// TwinCAT 3 PLC project PLCPro
// ProgramVersion: 3.1.4024.0
// libraries:
//   Tc2_Standard, * (Beckhoff Automation GmbH)
//   Tc2_System, * (Beckhoff Automation GmbH)
//   Tc2_Utilities, * (Beckhoff Automation GmbH)
//   Tc3_IotBase, * (Beckhoff Automation GmbH)
//   Tc3_JsonXml, * (Beckhoff Automation GmbH)
//   Tc3_Module, * (Beckhoff Automation GmbH)
// project tree:
//   / PlcTask.TcTTO
//   POUs/ MockServer.TcPOU, MAIN.TcPOU, EtonSmartBreaker.TcPOU, PostmanEco.TcPOU
// real-time tasks:
//   TASK PlcTask: cycle T#10ms, priority 20, ADS port 350

CONFIGURATION PLCPro
    RESOURCE PLC ON TwinCAT3
        TASK PlcTask(INTERVAL := T#10ms, PRIORITY := 20);
        PROGRAM MAIN WITH PlcTask : MAIN;
    END_RESOURCE
END_CONFIGURATION

// ---- POUs/MAIN.TcPOU
PROGRAM MAIN
VAR
	//Client
	//fbhttpClient : FB_IotHttpClient := (sHostName:='postman-echo.com',
	//							  	bKeepAlive:=TRUE, tConnectionTimeout:=T#10S);
									
	//Eton
	fbhttpClient : FB_IotHttpClient := (sHostName:='api.em.eaton.com',
								  	bKeepAlive:=TRUE, tConnectionTimeout:=T#10S);		
				
	//Get Request
	fbRequest : FB_IotHttpRequest;		
	state : (IDLE, SEND_REQUEST, WAIT_FOR_RESPONSE, READ_RESPONSE,ERROR,FORMATER);			
	sendGetRequest: BOOL;
	debugContent : STRING(511);
	fbJsonParser : FB_JsonDomParser;
	jsonDoc				: SJsonValue;
	jsonArgsMember				: SJsonValue;
	jsonFoo2 : SJsonValue;
	results : STRING;
	
	//JSON Formater
	fbJsonWriter         : FB_JsonSaxWriter;
	sendData                : STRING(2000);
	
END_VAR

//PostmanEco();
MockServer();
//EtonSmartBreaker();

END_PROGRAM

// ---- POUs/MockServer.TcPOU
PROGRAM MockServer
VAR
	//Mock Server
	fbhttpClient : FB_IotHttpClient := (sHostName:='4446f140-18dd-4b14-8279-3cc341a02b1e.mock.pstmn.io',
								  	bKeepAlive:=TRUE, tConnectionTimeout:=T#10S);		
				
	//Get Request
	fbRequest : FB_IotHttpRequest;		
	state : (IDLE, SEND_REQUEST, WAIT_FOR_RESPONSE, READ_RESPONSE,ERROR,HEADER);			
	sendGetRequest: BOOL;
	debugContent : STRING(511);
	fbJsonParser : FB_JsonDomParser;
	jsonDoc				: SJsonValue;
	jsonArgsMember				: SJsonValue;
	jsonMachineName : SJsonValue;
	results : STRING;
	
	//Header
	fbHeaderField : FB_IotHttpHeaderFieldMap;
END_VAR

// Init client parameters at startup
IF NOT fbhttpClient.bConfigured THEN 
	fbhttpClient.nHostPort:= 443; //80 for http  443 For https
	fbhttpClient.stTLS.bNoServerCertCheck:= TRUE;
END_IF

	
//Get Request
CASE state OF
	
	//Send Get Request
	IDLE:
		IF sendGetRequest THEN
			state := HEADER;
			sendGetRequest := FALSE;
		END_IF
	
	//Create Autorization Header File
	HEADER:
		fbHeaderField.AddField(sField:='Header1',sValue:='1',bAppendValue:=FALSE);
		fbHeaderField.AddField(sField:='Header2',sValue:='2',bAppendValue:=FALSE);
		state := SEND_REQUEST;
	
	//Send Get Request
	SEND_REQUEST:                                                                                      
		IF fbRequest.SendRequest(sUri:='/getmockdata', 
			fbClient:=fbhttpClient, eRequestType:=ETcIotHttpRequestType.HTTP_Get, 
				0, 0,fbHeader:=fbHeaderField ) THEN
			state := WAIT_FOR_RESPONSE;
		END_IF
	
	//Wait for Response
	WAIT_FOR_RESPONSE:

		IF NOT fbRequest.bBusy THEN
			IF fbRequest.bError THEN
				state := ERROR;
			ELSE
				state := READ_RESPONSE;
			END_IF
		END_IF
	
	//Read Response	
	READ_RESPONSE:
	
		//Get Response Content
		fbRequest.GetContent(pContent:= ADR(debugContent), nContentSize:= SIZEOF(debugContent), bSetNullTermination:= TRUE);
		
		//Check Status 
		IF fbRequest.nStatusCode >= 200 AND fbRequest.nStatusCode < 300 THEN
			jsonDoc:= fbRequest.GetJsonDomContent(fbJsonParser);
			
			//Check response has data in body
			IF jsonDoc <> 0 THEN
				
				//Check machine key is present 
				IF fbJsonParser.HasMember(jsonDoc, 'machine') THEN
					
					//Get Value for the specifed key
					jsonArgsMember:= fbJsonParser.FindMember(jsonDoc, 'machine');
					
					//Check wether data has an name key 	
					IF fbJsonParser.HasMember(jsonArgsMember, 'name')  THEN
						
						//Get Value for the specifed key
						jsonMachineName:= fbJsonParser.FindMember(jsonArgsMember, 'name');
						
							//Check data is a String
							IF fbJsonParser.IsString(jsonMachineName) THEN	
								
								//Get the Data 		
								results:= fbJsonParser.GetString(jsonMachineName);									
							END_IF
					END_IF
				END_IF
			END_IF
		END_IF
		state := IDLE;
		
	ERROR:
		//
		
		
END_CASE

//Cyclic Client 
fbhttpClient.Execute();

END_PROGRAM

// ---- POUs/EtonSmartBreaker.TcPOU
PROGRAM EtonSmartBreaker
VAR
	//Eaton Server
	fbhttpClient : FB_IotHttpClient := (sHostName:='api.em.eaton.com',
								  	bKeepAlive:=TRUE, tConnectionTimeout:=T#10S);		
	
	//Get Request
	fbRequest : FB_IotHttpRequest;		
	state : (IDLE, SEND_REQUEST, WAIT_FOR_RESPONSE, READ_RESPONSE,ERROR,ADD_HEADER);			
	sendGetRequest: BOOL;
	debugContent : STRING(2000);
	fbJsonParser : FB_JsonDomParser;
	jsonDoc				: SJsonValue;
	jsonArgsMember				: SJsonValue;
	jsonMachineName : SJsonValue;
	results : STRING;
	
	//Header
	fbHeaderField : FB_IotHttpHeaderFieldMap;
	sAuthoToken : STRING(2000);
END_VAR

// Init client parameters at startup
IF NOT fbhttpClient.bConfigured THEN 
	fbhttpClient.nHostPort:= 443; //80 for http  443 For https
	fbhttpClient.stTLS.bNoServerCertCheck:= TRUE;
END_IF

	
//Get Request
CASE state OF
	
	//Send Get Request
	IDLE: 
		IF sendGetRequest THEN
			state := ADD_HEADER;
			sendGetRequest := FALSE;
		END_IF
	
	//Create Autorization Header File
	ADD_HEADER:
		sAuthoToken := 'Bearer eyJraWQiOiJFZHViWGxfQVg2emd3R044b0dOa21VRUxRWHEyOUdOQzNJUjFrcFdtVGZBIiwiYWxnIjoiUlMyNTYifQ.eyJ2ZXIiOjEsImp0aSI6IkFULjhjYU5jckV2aU56UHBKNEk1bEQ2YVh0amxjVTJ2TG9xQ29wcmNWd0ExdVUiLCJpc3MiOiJodHRwczovL2lkLmVhdG9uLmNvbS9vYXV0aDIvYXVzOWQ4dnhlOFZNWTFod0M0eDciLCJhdWQiOiJhcGk6Ly9ibGMiLCJpYXQiOjE3Mjc5MzE0MjMsImV4cCI6MTcyNzkzNTAyMywiY2lkIjoiMG9hbTgzZHR2dVdnV1FTNjk0eDciLCJzY3AiOlsiY2xpZW50X2NyZWQiXSwiYWRvcHRlcmlkIjoiYjgzYjJlZjItMmJhZi1iZTEzLTNmOGItZGI3ZmQyNWYyMDE3Iiwic3ViIjoiMG9hbTgzZHR2dVdnV1FTNjk0eDciLCJibGNzYWlkIjoiMGEzYmVhYTctZTE1ZS00N2U1LTlhMmItY2ZjYjE3ZGU1ZDQ0IiwibmFtZSI6IiAifQ.00_Ss224pRcBLPLgnpvzWnFV0GmS_tGB9qeZJu8OeWvd7kSRdSMygCW7wede4vqgu5Ubb5BiEe9cokUyDZlxNh-5BjZUgMOYV3XZXAJ5Rhxdnk4yjf6ERhz2HZ8PuB8aCMRdxaAe6N6f_PemYtNiTWQ7DWPPc7aFGsk2gy1FRxRTvX5XlgX2cIQoJKBBEq6lzWZOUW8Jl9Aw2f90uQ6BSJRAfazYmr6yWAjuQoOGHQlXHmZxGf1fEm9NqKGUeh5tYEAE-YueOLzh__bxsjUHR1NJwBrpN3sa3_VFoNzfGEunkiQ1RyFZyzoUS3xEB2QbCjJTgo47z_0nJobPwB3EDg';
		fbHeaderField.AddField(sField:='Em-Api-Subscription-Key',sValue:='666585a90d81461da51fb9ed6fa14c7b',bAppendValue:=FALSE);
		fbHeaderField.AddField(sField:='Authorization',sValue:=sAuthoToken,bAppendValue:=FALSE);
		//fbHeaderField.AddField(sField:='Accept',sValue:='application/json',bAppendValue:=FALSE);
		//fbHeaderField.AddField(sField:='Content-Type',sValue:='application/json',bAppendValue:=FALSE);
		//fbHeaderField.AddField(sField:='Cache-Control',sValue:='no-cache',bAppendValue:=FALSE);
		//fbHeaderField.AddField(sField:='Connection',sValue:='keep-alive',bAppendValue:=FALSE);
		state := SEND_REQUEST;
	
	//Send Get Request
	SEND_REQUEST:                                                                             
		IF fbRequest.SendRequest(sUri:='/api/v1/devices/c595f832-81c8-44c9-ba4a-0b3c9b980dc4/breaker/remoteHandle/position', 
			fbClient:=fbhttpClient, eRequestType:=ETcIotHttpRequestType.HTTP_Get, 
				0, 0,fbHeader:=fbHeaderField ) THEN
			state := WAIT_FOR_RESPONSE;
		END_IF

	//Wait for Response
	WAIT_FOR_RESPONSE:

		IF NOT fbRequest.bBusy THEN
			IF fbRequest.bError THEN
				state := ERROR;
			ELSE
				state := READ_RESPONSE;
			END_IF
		END_IF
	
	//Read Response
	READ_RESPONSE:
	
		//Get Response Content
		fbRequest.GetContent(pContent:= ADR(debugContent), nContentSize:= SIZEOF(debugContent), bSetNullTermination:= TRUE);
		
		//Check Status 
		IF fbRequest.nStatusCode >= 200 AND fbRequest.nStatusCode < 300 THEN
			jsonDoc:= fbRequest.GetJsonDomContent(fbJsonParser);
			
			//Check response has data in body
			IF jsonDoc <> 0 THEN
				
				//Check data key is present 
				IF fbJsonParser.HasMember(jsonDoc, 'data') THEN
					
					//Get Value for the specifed key
					jsonArgsMember:= fbJsonParser.FindMember(jsonDoc, 'data');
					
					//Check wether data has an position key
					IF fbJsonParser.HasMember(jsonArgsMember, 'position')  THEN
						
						//Get Value for the specifed key
						jsonMachineName:= fbJsonParser.FindMember(jsonArgsMember, 'position');
							
							//Check data is a String
							IF fbJsonParser.IsString(jsonMachineName) THEN			

								//Get the Data 				
								results:= fbJsonParser.GetString(jsonMachineName);									
							END_IF
					END_IF
				END_IF
			END_IF
		END_IF
		
		state := IDLE;
		
	ERROR:
		//Error Handling 
		
		
END_CASE

//Cyclic Client 
fbhttpClient.Execute();

END_PROGRAM

// ---- POUs/PostmanEco.TcPOU
PROGRAM PostmanEco
VAR
	//Client
	fbhttpClient : FB_IotHttpClient := (sHostName:='postman-echo.com',
								  	bKeepAlive:=TRUE, tConnectionTimeout:=T#10S);
	//Get Request
	fbRequest : FB_IotHttpRequest;		
	state : (IDLE, SEND_REQUEST, WAIT_FOR_RESPONSE, READ_RESPONSE,ERROR,FORMATER);			
	sendGetRequest: BOOL;
	debugContent : STRING(511);
	fbJsonParser : FB_JsonDomParser;
	jsonDoc				: SJsonValue;
	jsonArgsMember				: SJsonValue;
	jsonFoo2 : SJsonValue;
	results : STRING;
	
	
END_VAR

// Init client parameters at startup
IF NOT fbhttpClient.bConfigured THEN 
	fbhttpClient.nHostPort:= 443; //80 for http  443 For https
	fbhttpClient.stTLS.bNoServerCertCheck:= TRUE;
END_IF

	
//Get Request
CASE state OF
	
	IDLE:
		IF sendGetRequest THEN
			state := SEND_REQUEST;
			sendGetRequest := FALSE;
		END_IF
		
	SEND_REQUEST:                                                                                      
		IF fbRequest.SendRequest(sUri:='/get?foo1=bar1&foo2=bar2', 
			fbClient:=fbhttpClient, eRequestType:=ETcIotHttpRequestType.HTTP_Get, 0, 0, 0) THEN
			state := WAIT_FOR_RESPONSE;
		END_IF

	WAIT_FOR_RESPONSE:
		IF NOT fbRequest.bBusy THEN
			IF fbRequest.bError THEN
				state := ERROR;
			ELSE
				state := READ_RESPONSE;
			END_IF
		END_IF
		
	READ_RESPONSE:
	
		fbRequest.GetContent(pContent:= ADR(debugContent), nContentSize:= SIZEOF(debugContent), bSetNullTermination:= TRUE);
		
		IF fbRequest.nStatusCode >= 200 AND fbRequest.nStatusCode < 300 THEN
			jsonDoc:= fbRequest.GetJsonDomContent(fbJsonParser);
			
			IF jsonDoc <> 0 THEN
				
				IF fbJsonParser.HasMember(jsonDoc, 'args') THEN
					jsonArgsMember:= fbJsonParser.FindMember(jsonDoc, 'args');
					
					IF fbJsonParser.HasMember(jsonArgsMember, 'foo2')  THEN
						jsonFoo2:= fbJsonParser.FindMember(jsonArgsMember, 'foo2');
						
							IF fbJsonParser.IsString(jsonFoo2) THEN							
								results:= fbJsonParser.GetString(jsonFoo2);									
							END_IF
					END_IF
				END_IF
			END_IF
		END_IF
		state := IDLE;
		
	ERROR:
		//
		
		
END_CASE

//Cyclic Client 
fbhttpClient.Execute();

END_PROGRAM
